// TwinCAT 3 PLC project IOLib
// ProgramVersion: 3.1.4023.0
// libraries:
//   Tc2_Standard, * (Beckhoff Automation GmbH)
//   Tc2_System, * (Beckhoff Automation GmbH)
//   Tc3_Module, * (Beckhoff Automation GmbH)
// project tree:
//   CAN/ FB_CANControl.TcPOU, ITF_CANControl.TcIO, ST_TxRxMessage.TcDUT, ST_TxRxQueue.TcDUT
//   EtherCAT/EtherCAT Devices/ DeviceInfo.TcDUT (not stored), DeviceState.TcDUT (not stored), EtherCATDeviceBase.TcPOU (not stored)
//   EtherCAT/EtherCAT Master/ EcMasterInputs.TcDUT, MasterDevState.TcDUT
//   EtherCAT/Tasks/ EcMasterConfDevices.TcPOU, EcMasterDeviceCount.TcPOU, EcMasterDeviceState.TcPOU, EcMasterFrameCount.TcPOU, EcMasterFrameStats.TcPOU, EcMasterGetAbnortalStateChange.TcPOU, EcMasterGetDeviceCRC.TcPOU, EcMasterGetDeviceId.TcPOU, EcMasterGetDeviceState.TcPOU, EcMasterProtocolError.TcPOU, EcMasterScanDevices.TcPOU, EcMasterState.TcPOU, IEcTask.TcIO, ITask.TcIO
//   EtherNetIP/ EtherNetIPDeviceBase.TcPOU, EtherNetIPMaster.TcPOU
//   Motion/RollerAxis/ EP7402_0xxx_Channel.TcPOU
//   Motion/RollerAxis/Structs/ DInputs.TcDUT, DOutputs.TcDUT, STMControl.TcDUT, STMInfoData.TcDUT, STMInputDevice.TcDUT, STMStatus.TcDUT, STMTargetVelocity.TcDUT
//   Motion/ServoAxis/ Exx72x1_DMC_Channel.TcPOU
//   Motion/ServoAxis/Structs/ DMC_Ins.TcDUT, DMC_Outs.TcDUT, DriveControl.TcDUT, DriveInputs.TcDUT, DriveOutputs.TcDUT, DriveStatus.TcDUT, PositioningControl.TcDUT, PositionStatus.TcDUT
//   Motion/StepperAxis/ Ex70x7_DMC_Channel.TcPOU
//   Motion/StepperAxis/Structs/ StartType.TcDUT, StepperENCControl.TcDUT, StepperENCStatus.TcDUT, StepperPOSControl.TcDUT, StepperPOSStatus.TcDUT, StepperSTMControl.TcDUT, StepperSTMStatus.TcDUT
//   / PlcTask.TcTTO
//   POUs/ MAIN.TcPOU
//   Profibus/ ProfibusDeviceBase.TcPOU, ProfibusMaster.TcPOU
//   ProfiNet/ ProfiNetDeviceBase.TcPOU, ProfiNetMaster.TcPOU

CONFIGURATION IOLib
    RESOURCE PLC ON TwinCAT3
        TASK PlcTask(INTERVAL := T#10ms, PRIORITY := 20);
        PROGRAM MAIN WITH PlcTask : MAIN;
    END_RESOURCE
END_CONFIGURATION

// ---- CAN/ST_TxRxMessage.TcDUT
{attribute 'pack_mode' := '1'} 
TYPE ST_TxRxMessage :
STRUCT
	dataLength : UINT;
	cobId : UDINT;
	data : ARRAY[0..7] OF BYTE;
END_STRUCT
END_TYPE

// ---- CAN/ST_TxRxQueue.TcDUT
TYPE ST_TxRxQueue :
STRUCT
	txCounter : UINT;
	rxCounter : UINT;
	noOfMessages : UINT;
	messages : ARRAY[0..9] OF ST_TxRxMessage;
END_STRUCT
END_TYPE

// ---- EtherCAT/EtherCAT Master/EcMasterInputs.TcDUT
TYPE EcMasterInputs :
STRUCT
	SlaveCount : UINT;
	DevState : UINT;
END_STRUCT
END_TYPE

// ---- EtherCAT/EtherCAT Master/MasterDevState.TcDUT
{attribute 'qualified_only'}
{attribute 'strict'}
TYPE MasterDevState :
(
	enum_member := 0
);
END_TYPE

// ---- Motion/RollerAxis/Structs/DInputs.TcDUT
TYPE DInputs :
STRUCT
	input1 : BOOL;
	input2 : BOOL;
	input3 : BOOL;
	input4 : BOOL;
	controlInput1 : BOOL;
	controlInput2 : BOOL;
	controlInput3 : BOOL;
	controlInput4 : BOOL;
END_STRUCT
END_TYPE

// ---- Motion/RollerAxis/Structs/DOutputs.TcDUT
TYPE DOutputs :
STRUCT
	output1 : BOOL;
	output2 : BOOL;
	output3 : BOOL;
	output4 : BOOL;
	controlOutput1 : BOOL;
	controlOutput2 : BOOL;
	controlOutput3 : BOOL;
	controlOutput4 : BOOL;
END_STRUCT
END_TYPE

// ---- Motion/RollerAxis/Structs/STMControl.TcDUT
TYPE STMControl :
STRUCT
	enable : BOOL;
	reset : BOOL;
	invertDirection : BOOL;
	brakeOutput : BOOL;
END_STRUCT
END_TYPE

// ---- Motion/RollerAxis/Structs/STMInfoData.TcDUT
TYPE STMInfoData :
STRUCT
	infoData1 : UINT;
	infoData2 : UINT;
	infoData3 : UINT;
END_STRUCT
END_TYPE

// ---- Motion/RollerAxis/Structs/STMInputDevice.TcDUT
TYPE STMInputDevice :
STRUCT
	deviceUnderVoltage : BOOL;
	deviceOverVoltage : BOOL;
	overTemperatureWarning : BOOL;
	overTemperatureError : BOOL;
	generalHWError : BOOL;
	chn1OpenLoad : BOOL;
	chn1ShortCircuit : BOOL;
	chn1MotorOverloadI2TWarning : BOOL;
	chn1MotorOverloadI2TError : BOOL;
	chn1AmplifierOverloadI2TWarning : BOOL;
	chn1AmplifierOverloadI2TError : BOOL;
	chn1InLimit : BOOL;
	chn1CommutationError : BOOL;
	chn2OpenLoad : BOOL;
	chn2ShortCircuit : BOOL;
	chn2MotorOverloadI2TWarning : BOOL;
	chn2MotorOverloadI2TError : BOOL;
	chn2AmplifierOverloadI2TWarning : BOOL;
	chn2AmplifierOverloadI2TError : BOOL;
	chn2InLimit : BOOL;
	chn2CommutationError : BOOL;
END_STRUCT
END_TYPE

// ---- Motion/RollerAxis/Structs/STMStatus.TcDUT
TYPE STMStatus :
STRUCT
	readyToEnable : BOOL;
	ready : BOOL;
	warning : BOOL;
	error : BOOL;
	movingPositive : BOOL;
	movingNegative : BOOL;
	txPDOToggle : BOOL;
END_STRUCT
END_TYPE

// ---- Motion/RollerAxis/Structs/STMTargetVelocity.TcDUT
TYPE STMTargetVelocity :
STRUCT
	velocity : INT;
	acceleration : UINT;
	deceleration : UINT;
END_STRUCT
END_TYPE

// ---- Motion/ServoAxis/Structs/DMC_Ins.TcDUT
TYPE DMC_Ins :
STRUCT
	DMC_Inputs : DriveInputs;
	DMC_POS_Status : PositionStatus;
	DMC_Drv_Status : DriveStatus;
END_STRUCT
END_TYPE

// ---- Motion/ServoAxis/Structs/DMC_Outs.TcDUT
TYPE DMC_Outs :
STRUCT
	DMC_DrvOuts : DriveOutputs;
	DMC_Drv_Ctrl : DriveControl;
	DMC_POS_Ctrl : PositioningControl;
END_STRUCT
END_TYPE

// ---- Motion/ServoAxis/Structs/DriveControl.TcDUT
TYPE DriveControl :
STRUCT
	Enable : BOOL;
	Reset : BOOL;
END_STRUCT
END_TYPE

// ---- Motion/ServoAxis/Structs/DriveInputs.TcDUT
TYPE DriveInputs :
STRUCT
	SetPosition : UDINT;
	SetVelocity : INT;
	ActualDriveTime : UDINT;
	ActualPositionLag : DINT;
	ActualVelocity : INT;
	ActualPosition : UDINT;
	ErrorId : UDINT;
	InputCycleCounter : USINT;
	LatchValue : UDINT;
	CyclicInfoData1 : INT;
	CyclicInforData2 : INT;
END_STRUCT
END_TYPE

// ---- Motion/ServoAxis/Structs/DriveOutputs.TcDUT
TYPE DriveOutputs :
STRUCT
	SetCounterValue : UDINT;
	TargetPosition : UDINT;
	TargetVelocity : INT;
	StartType : UINT;
	TargetAcceleration : UINT;
	TargetDeceleration : UINT;
END_STRUCT
END_TYPE

// ---- Motion/ServoAxis/Structs/DriveStatus.TcDUT
TYPE DriveStatus :
STRUCT
	ReadyToEnable : BOOL;
	Ready : BOOL;
	Warning : BOOL;
	Error : BOOL;
	MovingPositive : BOOL;
	MovingNegative : BOOL;
	DigitalInput1 : BOOL;
	DigitalInput2 : BOOL;
END_STRUCT
END_TYPE

// ---- Motion/ServoAxis/Structs/PositioningControl.TcDUT
TYPE PositioningControl :
STRUCT
	Execute : BOOL;
	EmergencyStop : BOOL;
END_STRUCT
END_TYPE

// ---- Motion/ServoAxis/Structs/PositionStatus.TcDUT
TYPE PositionStatus :
STRUCT
	Busy : BOOL;
	InTarget : BOOL;
	Warning : BOOL;
	Error : BOOL;
	Calibrated : BOOL;
	Accelerate : BOOL;
	Decelerate : BOOL;
	ReadyToExecute : BOOL;
END_STRUCT
END_TYPE

// ---- Motion/StepperAxis/Structs/StartType.TcDUT
{attribute 'qualified_only'}
{attribute 'strict'}
TYPE StartType :
(
	Absolute := 1,
	Relative := 2,
	VeloPositive := 3,
	VeloNegative := 4,
	Calibrate := 24576 
);
END_TYPE

// ---- Motion/StepperAxis/Structs/StepperENCControl.TcDUT
TYPE StepperENCControl :
STRUCT
	EnableLatchC : BOOL;
	EnableLatchPositiveEdge : BOOL;
	SetCounter : BOOL;
	EnableLatchNegativeEdge : BOOL;
	SetCounterValue : UDINT;
END_STRUCT
END_TYPE

// ---- Motion/StepperAxis/Structs/StepperENCStatus.TcDUT
TYPE StepperENCStatus :
STRUCT
	LatchCValid : BOOL;
	LatchExternalValid : BOOL;
	SetCounterDone : BOOL;
	CounterUnderflow : BOOL;
	CounterOverflow : BOOL;
	ExtrapolationStall : BOOL;
	StatusInputA : BOOL;
	StatusInputB : BOOL;
	StatusInputC : BOOL;
	StatusExternLatch : BOOL;
	SyncError : BOOL;
	TxPDOToggle : BOOL;
	CounterValue : UDINT;
	LatchValue : UDINT;
END_STRUCT
END_TYPE

// ---- Motion/StepperAxis/Structs/StepperPOSControl.TcDUT
TYPE StepperPOSControl :
STRUCT
	Execute : BOOL;
	EmergencyStop : BOOL;
	TargetPosition : UDINT;
	Velocity : INT;
	StartType : UINT;
	Acceleration : UINT;
	Deceleration : UINT;
END_STRUCT
END_TYPE

// ---- Motion/StepperAxis/Structs/StepperPOSStatus.TcDUT
TYPE StepperPOSStatus :
STRUCT
	Busy : BOOL;
	InTarget : BOOL;
	Warning : BOOL;
	Error : BOOL;
	Calibrated : BOOL;
	Accelerate : BOOL;
	Decelerate : BOOL;
	ReadyToExecute : BOOL;
	ActualPosition : UDINT;
	ActualVelocity : INT;
	ActualDriveTime : UDINT;
END_STRUCT
END_TYPE

// ---- Motion/StepperAxis/Structs/StepperSTMControl.TcDUT
TYPE StepperSTMControl :
STRUCT
	Enable : BOOL;
	Reset : BOOL;
	ReduceTorque : BOOL;
	DigitalOutput1 : BOOL;
END_STRUCT
END_TYPE

// ---- Motion/StepperAxis/Structs/StepperSTMStatus.TcDUT
TYPE StepperSTMStatus :
STRUCT
	ReadyToEnable : BOOL;
	Ready : BOOL;
	Warning : BOOL;
	Error : BOOL;
	MovingPositive : BOOL;
	MovingNegative : BOOL;
	MotorStall : BOOL;
	DigitalInput1 : BOOL;
	DigitalInput2 : BOOL;
	SyncError : BOOL;
	TxPDOToggle : BOOL;
END_STRUCT
END_TYPE

// ---- CAN/ITF_CANControl.TcIO
INTERFACE ITF_CANControl

METHOD M_GetMessage : BOOL
VAR_INPUT
END_VAR
END_METHOD

METHOD M_PushMessage : BOOL
VAR_INPUT
	messageSend : ST_TxRxMessage;
END_VAR
END_METHOD

END_INTERFACE

// ---- EtherCAT/Tasks/IEcTask.TcIO
INTERFACE IEcTask EXTENDS ITask

PROPERTY NetID : amsnetid
GET
END_GET
SET
END_SET
END_PROPERTY

END_INTERFACE

// ---- EtherCAT/Tasks/ITask.TcIO
INTERFACE ITask

METHOD Abort : BOOL
VAR_INPUT
END_VAR
END_METHOD

PROPERTY Busy : bool
GET
END_GET
END_PROPERTY

PROPERTY Done : bool
GET
END_GET
END_PROPERTY

PROPERTY Error : bool
GET
END_GET
END_PROPERTY

METHOD Execute : BOOL
VAR_INPUT
END_VAR
END_METHOD

END_INTERFACE

// ---- POUs/MAIN.TcPOU
PROGRAM MAIN
VAR
END_VAR

END_PROGRAM

// ---- CAN/FB_CANControl.TcPOU
FUNCTION_BLOCK PUBLIC FB_CANControl IMPLEMENTS ITF_CANControl
VAR_INPUT
END_VAR
VAR_OUTPUT
END_VAR
VAR
	rxQueue AT%I* : ST_TxRxQueue;
	txQueue AT%Q* : ST_TxRxQueue;
	i : INT;
	messageRecieved : ST_TxRxMessage;
END_VAR

IF rxQueue.rxCounter <> txQueue.rxCounter THEN
	//if we have recieved a message rxCounter is incremented by interface
	M_GetMessage();
END_IF

METHOD PUBLIC M_GetMessage : BOOL
VAR_INPUT
END_VAR
FOR i := 0 TO rxQueue.noOfMessages DO
	messageRecieved := rxQueue.messages[i];
END_FOR
txQueue.rxCounter := rxQueue.rxCounter;
END_METHOD

METHOD PUBLIC M_PushMessage : BOOL
VAR_INPUT
	messageSend : ST_TxRxMessage;
END_VAR
IF txQueue.txCounter = rxQueue.TxCounter THEN
	FOR i:=0 TO 1 DO
		txQueue.messages[i] := messageSend;
	End_for
	txQueue.noOfMessages := 1;
	txQueue.TxCounter := rxQueue.TxCounter + 1;
END_IF
END_METHOD

END_FUNCTION_BLOCK

// ---- EtherCAT/Tasks/EcMasterConfDevices.TcPOU
FUNCTION_BLOCK EcMasterConfDevices IMPLEMENTS IEcTask
VAR_INPUT
END_VAR
VAR_OUTPUT
END_VAR
VAR
	iState : INT;
	masterConfDevices : Tc2_EtherCAT.FB_EcGetConfSlaves;
	_confDevices : ARRAY[0..Tc2_EtherCAT.EC_MAX_SLAVES] OF Tc2_EtherCAT.ST_EcSlaveConfigData;
	_execute: BOOL;
	_done: BOOL;
	_busy: BOOL;	
	_error: BOOL;
	_netId: AMSNETID;
END_VAR

CASE iState OF
	0:
		IF _execute THEN
			_done := FALSE;
			_busy := TRUE;
			_error := FALSE;
			masterConfDevices.bExecute := TRUE;
			IF masterConfDevices.bBusy THEN
				iState := 10;
				_execute := FALSE;
			END_IF
		END_IF
	10:
		IF NOT masterConfDevices.bBusy THEN
			IF NOT masterConfDevices.bError THEN
				_done := TRUE;
			ELSE
				_error := TRUE;
			END_IF
			_busy := FALSE;
			masterConfDevices.bExecute := FALSE;
			iState := 0;
		END_IF
END_CASE

masterConfDevices(sNetId := Tc2_System.F_CreateAmsNetId(nIds := NetId), 
					pArrEcConfSlaveInfo := ADR(_confDevices), 
					cbBufLen := SIZEOF(_confDevices));

{warning 'add method implementation '}
METHOD Abort : BOOL
masterConfDevices.bExecute := FALSE;
_busy := FALSE;
_execute := FALSE;
Abort := TRUE;
iState := 0;
END_METHOD

{warning 'add property implementation'}
PROPERTY Busy : BOOL
GET
Busy := _busy;
END_GET
END_PROPERTY

PROPERTY ConfiguredDevices : reference to array[0..Ec_Max_slaves] of St_ecslaveconfigdata
GET
ConfiguredDevices REF= _confDevices;
END_GET
END_PROPERTY

{warning 'add property implementation'}
PROPERTY Done : BOOL
GET
Done := _done;
END_GET
END_PROPERTY

{warning 'add property implementation'}
PROPERTY Error : BOOL
GET
Error := _error;
END_GET
END_PROPERTY

{warning 'add method implementation '}
METHOD Execute : BOOL
IF NOT masterConfDevices.bBusy THEN
	Execute := _execute := true;
END_IF
END_METHOD

{warning 'add property implementation'}
PROPERTY NetID : amsnetid
GET
NetID := _netId;
END_GET
SET
_netId := NetID;
END_SET
END_PROPERTY

PROPERTY NumberConfDevices : udint
GET
NumberConfDevices := masterConfDevices.nSlaves;
END_GET
END_PROPERTY

END_FUNCTION_BLOCK

// ---- EtherCAT/Tasks/EcMasterDeviceCount.TcPOU
FUNCTION_BLOCK PUBLIC EcMasterDeviceCount IMPLEMENTS IEcTask
VAR_INPUT
END_VAR
VAR_OUTPUT
END_VAR
VAR
	iState : INT;
	masterDeviceCount : Tc2_EtherCAT.FB_EcGetSlaveCount;
	_execute: BOOL;
	_done: BOOL;
	_busy: BOOL;
	_error: BOOL;
	_netId: AMSNETID;
END_VAR

CASE iState OF
	0:
		IF _execute THEN
			_done := FALSE;
			_busy := TRUE;
			_error := FALSE;
			masterDeviceCount.bExecute := TRUE;
			IF masterDeviceCount.bBusy THEN
				iState := 10;
				_execute := false;
			END_IF
		END_IF
	10:
		IF NOT masterDeviceCount.bBusy THEN
			IF NOT masterDeviceCount.bError THEN
				_done := TRUE;
			ELSE
				_error := TRUE;
			END_IF
			_busy := FALSE;
			masterDeviceCount.bExecute := FALSE;
			iState := 0;
		END_IF
END_CASE

masterDeviceCount(sNetId := Tc2_System.F_CreateAmsNetId(nIds := NetId));

{warning 'add method implementation '}
METHOD Abort : BOOL
masterDeviceCount.bExecute := FALSE;
_busy := FALSE;
_execute := FALSE;
Abort := TRUE;
iState := 0;
END_METHOD

{warning 'add property implementation'}
PROPERTY Busy : BOOL
GET
Busy := _busy;
END_GET
END_PROPERTY

{warning 'add property implementation'}
PROPERTY Done : BOOL
GET
Done := _done;
END_GET
END_PROPERTY

{warning 'add property implementation'}
PROPERTY Error : BOOL
GET
Error := _error;
END_GET
END_PROPERTY

METHOD Execute : BOOL
VAR_INPUT
END_VAR
IF NOT Busy THEN
	Execute := _execute := TRUE;
END_IF
END_METHOD

{warning 'add property implementation'}
PROPERTY NetID : amsnetid
GET
NetID := _netId;
END_GET
SET
_netId := NetID;
END_SET
END_PROPERTY

PROPERTY NumberDevices : uint
GET
NumberDevices := masterDeviceCount.nSlaves;
END_GET
END_PROPERTY

END_FUNCTION_BLOCK

// ---- EtherCAT/Tasks/EcMasterDeviceState.TcPOU
FUNCTION_BLOCK EcMasterDeviceState IMPLEMENTS IEcTask
VAR_INPUT
END_VAR
VAR_OUTPUT
END_VAR
VAR
	iState : INT;
	masterDeviceState : Tc2_EtherCAT.FB_EcGetMasterDevState;
	_execute: BOOL;
	_done: BOOL;
	_busy: BOOL;
	_error: BOOL;
	_netId: AMSNETID;
END_VAR

CASE iState OF
	0:
		IF _execute THEN
			_done := FALSE;
			_busy := TRUE;
			_error := FALSE;
			masterDeviceState.bExecute := TRUE;
			IF masterDeviceState.bBusy THEN
				iState := 10;
				_execute := false;
			END_IF
		END_IF
	10:
		IF NOT masterDeviceState.bBusy THEN
			IF NOT masterDeviceState.bError THEN
				_done := TRUE;
			ELSE
				_error := TRUE;
			END_IF
			_busy := FALSE;
			masterDeviceState.bExecute := FALSE;
			iState := 0;
		END_IF
END_CASE

masterDeviceState(sNetId := Tc2_System.F_CreateAmsNetId(nIds := NetId));

{warning 'add method implementation '}
METHOD Abort : BOOL
masterDeviceState.bExecute := FALSE;
_busy := FALSE;
_execute := FALSE;
Abort := TRUE;
iState := 0;
END_METHOD

{warning 'add property implementation'}
PROPERTY Busy : BOOL
GET
Busy := _busy;
END_GET
END_PROPERTY

{warning 'add property implementation'}
PROPERTY Done : BOOL
GET
Done := _done;
END_GET
END_PROPERTY

{warning 'add property implementation'}
PROPERTY Error : BOOL
GET
Error := _error;
END_GET
END_PROPERTY

{warning 'add method implementation '}
METHOD Execute : BOOL
IF NOT masterDeviceState.bBusy THEN
	Execute := _execute := true;
END_IF
END_METHOD

PROPERTY MasterDevState : word
GET
MasterDevState := masterDeviceState.nDevState;
END_GET
END_PROPERTY

{warning 'add property implementation'}
PROPERTY NetID : amsnetid
GET
NetID := _netId;
END_GET
SET
_netId := NetID;
END_SET
END_PROPERTY

END_FUNCTION_BLOCK

// ---- EtherCAT/Tasks/EcMasterFrameCount.TcPOU
FUNCTION_BLOCK EcMasterFrameCount IMPLEMENTS IEcTask
VAR_INPUT
END_VAR
VAR_OUTPUT
END_VAR
VAR
	iState : INT;
	masterFrameCount : Tc2_EtherCAT.FB_EcMasterFrameCount;
	_execute: BOOL;
	_done: BOOL;
	_busy: BOOL;
	_error: BOOL;
	_netId: AMSNETID;
END_VAR

CASE iState OF
	0:
		IF _execute THEN
			_done := FALSE;
			_busy := TRUE;
			_error := FALSE;
			masterFrameCount.bExecute := TRUE;
			IF masterFrameCount.bBusy THEN
				iState := 10;
				_execute := false;
			END_IF
		END_IF
	10:
		IF NOT masterFrameCount.bBusy THEN
			IF NOT masterFrameCount.bError THEN
				_done := TRUE;
			ELSE
				_error := TRUE;
			END_IF
			_busy := FALSE;
			masterFrameCount.bExecute := FALSE;
			iState := 0;
		END_IF
END_CASE

masterFrameCount(sNetId := Tc2_System.F_CreateAmsNetId(nIds := NetId));

{warning 'add method implementation '}
METHOD Abort : BOOL
masterFrameCount.bExecute := FALSE;
_busy := FALSE;
_execute := FALSE;
Abort := TRUE;
iState := 0;
END_METHOD

{warning 'add property implementation'}
PROPERTY Busy : BOOL
GET
Busy := _busy;
END_GET
END_PROPERTY

{warning 'add property implementation'}
PROPERTY Done : BOOL
GET
Done := _done;
END_GET
END_PROPERTY

{warning 'add property implementation'}
PROPERTY Error : BOOL
GET
Error := _error;
END_GET
END_PROPERTY

{warning 'add method implementation '}
METHOD Execute : BOOL
IF NOT masterFrameCount.bBusy THEN
	Execute := _execute := True;
END_IF
END_METHOD

PROPERTY FrameNumber : UDINT
GET
FrameNumber := masterFrameCount.nFrames;
END_GET
END_PROPERTY

{warning 'add property implementation'}
PROPERTY NetID : amsnetid
GET
NetID := _netId;
END_GET
SET
_netId := NetID;
END_SET
END_PROPERTY

END_FUNCTION_BLOCK

// ---- EtherCAT/Tasks/EcMasterFrameStats.TcPOU
FUNCTION_BLOCK PUBLIC EcMasterFrameStats IMPLEMENTS IEcTask
VAR_INPUT
END_VAR
VAR_OUTPUT
END_VAR
VAR
	iState : INT;
	masterFrameStats : Tc2_EtherCAT.FB_EcMasterFrameStatistic;
	_execute: BOOL;
	_done: BOOL;
	_busy: BOOL;
	_error: BOOL;
	_netId: AMSNETID;
END_VAR

CASE iState OF
	0:
		IF _execute THEN
			_done := FALSE;
			_busy := TRUE;
			_error := FALSE;
			masterFrameStats.bExecute := TRUE;
			IF masterFrameStats.bBusy THEN
				iState := 10;
				_execute := false;
			END_IF
		END_IF
	10:
		IF NOT masterFrameStats.bBusy THEN
			IF NOT masterFrameStats.bError THEN
				_done := TRUE;
			ELSE
				_error := TRUE;
			END_IF
			_busy := FALSE;
			masterFrameStats.bExecute := FALSE;
			iState := 0;
		END_IF
END_CASE

masterFrameStats(sNetId := Tc2_System.F_CreateAmsNetId(nIds := NetId));

{warning 'add method implementation '}
METHOD Abort : BOOL
masterFrameStats.bExecute := FALSE;
_busy := FALSE;
_execute := FALSE;
Abort := TRUE;
iState := 0;
END_METHOD

{warning 'add property implementation'}
PROPERTY Busy : BOOL
GET
Busy := _busy;
END_GET
END_PROPERTY

{warning 'add property implementation'}
PROPERTY Done : BOOL
GET
Done := _done;
END_GET
END_PROPERTY

{warning 'add property implementation'}
PROPERTY Error : BOOL
GET
Error := _error;
END_GET
END_PROPERTY

METHOD Execute : BOOL
VAR_INPUT
END_VAR
IF NOT Busy THEN
	Execute := _execute := TRUE;
END_IF
END_METHOD

PROPERTY FramesPerSecond  : LREAL
GET
FramesPerSecond := masterFrameStats.fFramesPerSecond;
END_GET
END_PROPERTY

PROPERTY LostFrames : UDINT
GET
LostFrames := masterFrameStats.nLostFrames;
END_GET
END_PROPERTY

PROPERTY LostQueuedFrames : udint
GET
LostQueuedFrames := masterFrameStats.nLostQueuedFrames;
END_GET
END_PROPERTY

{warning 'add property implementation'}
PROPERTY NetID : amsnetid
GET
NetID := _netId;
END_GET
SET
_netId := NetID;
END_SET
END_PROPERTY

PROPERTY QueuedFramesPerSecond : lreal
GET
QueuedFramesPerSecond := masterFrameStats.fQueuedFramesPerSecond;
END_GET
END_PROPERTY

END_FUNCTION_BLOCK

// ---- EtherCAT/Tasks/EcMasterGetAbnortalStateChange.TcPOU
FUNCTION_BLOCK EcMasterGetAbnortalStateChange IMPLEMENTS IEcTask
VAR_INPUT
END_VAR
VAR_OUTPUT
END_VAR
VAR
	iState : INT;
	masterAbnormalStateChanges : Tc2_EtherCAT.FB_EcGetAllSlaveAbnormalStateChanges;
	_abnormalStates : ARRAY[0..Tc2_EtherCAT.EC_MAX_SLAVES] OF UDINT;
	_execute: BOOL;
	_done: BOOL;
	_busy: BOOL;
	_error: BOOL;
	_netId: AMSNETID;
END_VAR

CASE iState OF
	0:
		IF _execute THEN
			_done := FALSE;
			_busy := TRUE;
			_error := FALSE;
			masterAbnormalStateChanges.bExecute := TRUE;
			IF masterAbnormalStateChanges.bBusy THEN
				iState := 10;
				_execute := false;
			END_IF
		END_IF
	10:
		IF NOT masterAbnormalStateChanges.bBusy THEN
			IF NOT masterAbnormalStateChanges.bError THEN
				_done := TRUE;
			ELSE
				_error := TRUE;
			END_IF
			_busy := FALSE;
			masterAbnormalStateChanges.bExecute := FALSE;
			iState := 0;
		END_IF
END_CASE

masterAbnormalStateChanges(sNetId := Tc2_System.F_CreateAmsNetId(nIds := NetId),
							pAddrBuf := ADR(_abnormalStates),
							cbBufLen := SIZEOF(_abnormalStates));

PROPERTY AbnormalStateChanges : reference to array[0..EC_MAX_Slaves] of udint
GET
AbnormalStateChanges REF= _abnormalStates;
END_GET
END_PROPERTY

{warning 'add method implementation '}
METHOD Abort : BOOL
masterAbnormalStateChanges.bExecute := FALSE;
_busy := FALSE;
_execute := FALSE;
Abort := TRUE;
iState := 0;
END_METHOD

{warning 'add property implementation'}
PROPERTY Busy : BOOL
GET
Busy := _busy;
END_GET
END_PROPERTY

{warning 'add property implementation'}
PROPERTY Done : BOOL
GET
Done := _done;
END_GET
END_PROPERTY

{warning 'add property implementation'}
PROPERTY Error : BOOL
GET
Error := _error;
END_GET
END_PROPERTY

{warning 'add method implementation '}
METHOD Execute : BOOL
IF NOT masterAbnormalStateChanges.bBusy THEN
	Execute := _execute := true;
END_IF
END_METHOD

{warning 'add property implementation'}
PROPERTY NetID : amsnetid
GET
NetID := _netId;
END_GET
SET
_netId := NetID;
END_SET
END_PROPERTY

END_FUNCTION_BLOCK

// ---- EtherCAT/Tasks/EcMasterGetDeviceCRC.TcPOU
FUNCTION_BLOCK EcMasterGetDeviceCRC IMPLEMENTS IEcTask
VAR_INPUT
END_VAR
VAR_OUTPUT
END_VAR
VAR
	iState : INT;
	getDeviceCRC : Tc2_EtherCAT.FB_EcGetSlaveCrcErrorEx;
	_execute: BOOL;
	_done: BOOL;
	_busy: BOOL;
	_error: BOOL;
	_netId: AMSNETID;
END_VAR

CASE iState OF
	0:
		IF _execute THEN
			_done := FALSE;
			_busy := TRUE;
			_error := FALSE;
			getDeviceCRC.bExecute := TRUE;
			IF getDeviceCRC.bBusy THEN
				iState := 10;
				_execute := false;
			END_IF
		END_IF
	10:
		IF NOT getDeviceCRC.bBusy THEN
			IF NOT getDeviceCRC.bError THEN
				_done := TRUE;
			ELSE
				_error := TRUE;
			END_IF
			_busy := FALSE;
			getDeviceCRC.bExecute := FALSE;
			iState := 0;
		END_IF
END_CASE

getDeviceCRC(sNetId := Tc2_System.F_CreateAmsNetId(nIds := NetId));

{warning 'add method implementation '}
METHOD Abort : BOOL
getDeviceCRC.bExecute := FALSE;
_busy := FALSE;
_execute := FALSE;
Abort := TRUE;
iState := 0;
END_METHOD

{warning 'add property implementation'}
PROPERTY Busy : BOOL
GET
Busy := _busy;
END_GET
END_PROPERTY

PROPERTY DeviceAddr : uint
GET
DeviceAddr := getDeviceCRC.nSlaveAddr;
END_GET
SET
getDeviceCRC.nSlaveAddr := DeviceAddr;
END_SET
END_PROPERTY

PROPERTY DeviceCRC :  ST_EcCrcErrorEx
GET
DeviceCRC := getDeviceCRC.crcError;
END_GET
END_PROPERTY

{warning 'add property implementation'}
PROPERTY Done : BOOL
GET
Done := _done;
END_GET
END_PROPERTY

{warning 'add property implementation'}
PROPERTY Error : BOOL
GET
Error := _error;
END_GET
END_PROPERTY

{warning 'add method implementation '}
METHOD Execute : BOOL
IF NOT getDeviceCRC.bBusy THEN
	Execute := _execute := true;
END_IF
END_METHOD

{warning 'add property implementation'}
PROPERTY NetID : amsnetid
GET
NetID := _netId;
END_GET
SET
_netId := NetID;
END_SET
END_PROPERTY

END_FUNCTION_BLOCK

// ---- EtherCAT/Tasks/EcMasterGetDeviceId.TcPOU
FUNCTION_BLOCK EcMasterGetDeviceId IMPLEMENTS IEcTask
VAR_INPUT
END_VAR
VAR_OUTPUT
END_VAR
VAR
	iState : INT;
	getDeviceIdentity : Tc2_EtherCAT.FB_EcGetSlaveIdentity;
	_execute: BOOL;
	_done: BOOL;
	_busy: BOOL;
	_error: BOOL;
	_netId: AMSNETID;
END_VAR

CASE iState OF
	0:
		IF _execute THEN
			_done := FALSE;
			_busy := TRUE;
			_error := FALSE;
			getDeviceIdentity.bExecute := TRUE;
			IF getDeviceIdentity.bBusy THEN
				iState := 10;
				_execute := false;
			END_IF
		END_IF
	10:
		IF NOT getDeviceIdentity.bBusy THEN
			IF NOT getDeviceIdentity.bError THEN
				_done := TRUE;
			ELSE
				_error := TRUE;
			END_IF
			_busy := FALSE;
			getDeviceIdentity.bExecute := FALSE;
			iState := 0;
		END_IF
END_CASE

getDeviceIdentity(sNetId := Tc2_System.F_CreateAmsNetId(nIds := NetId));

{warning 'add method implementation '}
METHOD Abort : BOOL
getDeviceIdentity.bExecute := FALSE;
_busy := FALSE;
_execute := FALSE;
Abort := TRUE;
iState := 0;
END_METHOD

{warning 'add property implementation'}
PROPERTY Busy : BOOL
GET
Busy := _busy;
END_GET
END_PROPERTY

PROPERTY DeviceAddr : uint
GET
DeviceAddr := getDeviceIdentity.nSlaveAddr;
END_GET
SET
getDeviceIdentity.nSlaveAddr := DeviceAddr;
END_SET
END_PROPERTY

PROPERTY DeviceIdentity : ST_EcSlaveIdentity
GET
DeviceIdentity := getDeviceIdentity.identity;
END_GET
END_PROPERTY

{warning 'add property implementation'}
PROPERTY Done : BOOL
GET
Done := _done;
END_GET
END_PROPERTY

{warning 'add property implementation'}
PROPERTY Error : BOOL
GET
Error := _error;
END_GET
END_PROPERTY

{warning 'add method implementation '}
METHOD Execute : BOOL
IF NOT getDeviceIdentity.bBusy THEN
	Execute := _execute := true;
END_IF
END_METHOD

{warning 'add property implementation'}
PROPERTY NetID : amsnetid
GET
NetID := _netId;
END_GET
SET
_netId := NetID;
END_SET
END_PROPERTY

END_FUNCTION_BLOCK

// ---- EtherCAT/Tasks/EcMasterGetDeviceState.TcPOU
FUNCTION_BLOCK EcMasterGetDeviceState IMPLEMENTS IEcTask
VAR_INPUT
END_VAR
VAR_OUTPUT
END_VAR
VAR
	iState : INT;
	getDeviceState : Tc2_EtherCAT.FB_EcGetSlaveState;
	_execute: BOOL;
	_done: BOOL;
	_busy: BOOL;
	_error: BOOL;
	_netId: AMSNETID;
END_VAR

CASE iState OF
	0:
		IF _execute THEN
			_done := FALSE;
			_busy := TRUE;
			_error := FALSE;
			getDeviceState.bExecute := TRUE;
			IF getDeviceState.bBusy THEN
				iState := 10;
				_execute := false;
			END_IF
		END_IF
	10:
		IF NOT getDeviceState.bBusy THEN
			IF NOT getDeviceState.bError THEN
				_done := TRUE;
			ELSE
				_error := TRUE;
			END_IF
			_busy := FALSE;
			getDeviceState.bExecute := FALSE;
			iState := 0;
		END_IF
END_CASE

getDeviceState(sNetId := Tc2_System.F_CreateAmsNetId(nIds := NetId));

{warning 'add method implementation '}
METHOD Abort : BOOL
getDeviceState.bExecute := FALSE;
_busy := FALSE;
_execute := FALSE;
Abort := TRUE;
iState := 0;
END_METHOD

{warning 'add property implementation'}
PROPERTY Busy : BOOL
GET
Busy := _busy;
END_GET
END_PROPERTY

PROPERTY DeviceAddr : uint
GET
DeviceAddr := getDeviceState.nSlaveAddr;
END_GET
SET
getDeviceState.nSlaveAddr := DeviceAddr;
END_SET
END_PROPERTY

PROPERTY DeviceState : ST_EcSlaveState
GET
DeviceState := getDeviceState.state;
END_GET
END_PROPERTY

{warning 'add property implementation'}
PROPERTY Done : BOOL
GET
Done := _done;
END_GET
END_PROPERTY

{warning 'add property implementation'}
PROPERTY Error : BOOL
GET
Error := _error;
END_GET
END_PROPERTY

{warning 'add method implementation '}
METHOD Execute : BOOL
IF NOT getDeviceState.bBusy THEN
	Execute := _execute := true;
END_IF
END_METHOD

{warning 'add property implementation'}
PROPERTY NetID : amsnetid
GET
NetID := _netId;
END_GET
SET
_netId := NetID;
END_SET
END_PROPERTY

END_FUNCTION_BLOCK

// ---- EtherCAT/Tasks/EcMasterProtocolError.TcPOU
FUNCTION_BLOCK EcMasterProtocolError IMPLEMENTS IEcTask
VAR_INPUT
END_VAR
VAR_OUTPUT
END_VAR
VAR
	iState : INT;
	masterProtocolErr : Tc2_EtherCAT.FB_EcGetLastProtErrInfo;
	_execute: BOOL;
	_done: BOOL;
	_busy: BOOL;
	_error: BOOL;
	_netId: AMSNETID;
END_VAR

CASE iState OF
	0:
		IF _execute THEN
			_done := FALSE;
			_busy := TRUE;
			_error := FALSE;
			masterProtocolErr.bExecute := TRUE;
			IF masterProtocolErr.bBusy THEN
				iState := 10;
				_execute := false;
			END_IF
		END_IF
	10:
		IF NOT masterProtocolErr.bBusy THEN
			IF NOT masterProtocolErr.bError THEN
				_done := TRUE;
			ELSE
				_error := TRUE;
			END_IF
			_busy := FALSE;
			masterProtocolErr.bExecute := FALSE;
			iState := 0;
		END_IF
END_CASE

masterProtocolErr(sNetId := Tc2_System.F_CreateAmsNetId(nIds := NetId));

{warning 'add method implementation '}
METHOD Abort : BOOL
masterProtocolErr.bExecute := FALSE;
_busy := FALSE;
_execute := FALSE;
Abort := TRUE;
iState := 0;
END_METHOD

{warning 'add property implementation'}
PROPERTY Busy : BOOL
GET
Busy := _busy;
END_GET
END_PROPERTY

PROPERTY DeviceAddr : uint
GET
DeviceAddr := masterProtocolErr.nSlaveAddr;
END_GET
SET
masterProtocolErr.nSlaveAddr := DeviceAddr;
END_SET
END_PROPERTY

{warning 'add property implementation'}
PROPERTY Done : BOOL
GET
Done := _done;
END_GET
END_PROPERTY

{warning 'add property implementation'}
PROPERTY Error : BOOL
GET
Error := _error;
END_GET
END_PROPERTY

{warning 'add method implementation '}
METHOD Execute : BOOL
IF NOT masterProtocolErr.bBusy THEN
	Execute := _execute := TRUE;
END_IF
END_METHOD

PROPERTY LastProtocolError : ST_EcLastProtErrInfo
GET
LastProtocolError := masterProtocolErr.info;
END_GET
END_PROPERTY

{warning 'add property implementation'}
PROPERTY NetID : amsnetid
GET
NetID := _netId;
END_GET
SET
_netId := NetID;
END_SET
END_PROPERTY

PROPERTY ProtocolType : E_EcMbxProtType
GET
ProtocolType := masterProtocolErr.eProtocol;
END_GET
SET
masterProtocolErr.eProtocol := ProtocolType;
END_SET
END_PROPERTY

END_FUNCTION_BLOCK

// ---- EtherCAT/Tasks/EcMasterScanDevices.TcPOU
FUNCTION_BLOCK EcMasterScanDevices IMPLEMENTS IEcTask
VAR_INPUT
END_VAR
VAR_OUTPUT
END_VAR
VAR
	iState : INT;
	masterScanDevices : Tc2_EtherCAT.FB_EcGetScannedSlaves;
	_scanDevices : ARRAY[0..Tc2_EtherCAT.EC_MAX_SLAVES] OF Tc2_EtherCAT.ST_EcSlaveScannedData;
	_execute: BOOL;
	_done: BOOL;
	_busy: BOOL;
	_error: BOOL;
	_netId: AMSNETID;
END_VAR

CASE iState OF
	0:
		IF _execute THEN
			_done := FALSE;
			_busy := TRUE;
			_error := FALSE;
			masterScanDevices.bExecute := TRUE;
			IF masterScanDevices.bBusy THEN
				iState := 10;
				_execute := false;
			END_IF
		END_IF
	10:
		IF NOT masterScanDevices.bBusy THEN
			IF NOT masterScanDevices.bError THEN
				_done := TRUE;
			ELSE
				_error := TRUE;
			END_IF
			_busy := FALSE;
			masterScanDevices.bExecute := FALSE;
			iState := 0;
		END_IF
END_CASE

masterScanDevices(sNetId := Tc2_System.F_CreateAmsNetId(nIds := NetId), 
					pArrEcScannedSlaveInfo := ADR(_scanDevices), 
					cbBufLen := SIZEOF(_scanDevices));

{warning 'add method implementation '}
METHOD Abort : BOOL
masterScanDevices.bExecute := FALSE;
_busy := FALSE;
_execute := FALSE;
Abort := TRUE;
iState := 0;
END_METHOD

{warning 'add property implementation'}
PROPERTY Busy : BOOL
GET
Busy := _busy;
END_GET
END_PROPERTY

{warning 'add property implementation'}
PROPERTY Done : BOOL
GET
Done := _done;
END_GET
END_PROPERTY

{warning 'add property implementation'}
PROPERTY Error : BOOL
GET
Error := _error;
END_GET
END_PROPERTY

{warning 'add method implementation '}
METHOD Execute : BOOL
IF NOT masterScanDevices.bBusy THEN
	Execute := _execute := true;
END_IF
END_METHOD

{warning 'add property implementation'}
PROPERTY NetID : amsnetid
GET
NetID := _netId;
END_GET
SET
_netId := NetID;
END_SET
END_PROPERTY

PROPERTY NumberScanDevices : udint
GET
NumberScanDevices := masterScanDevices.nSlaves;
END_GET
END_PROPERTY

PROPERTY ScannedDevices : reference to array[0..EC_MAX_Slaves] of ST_EcSlaveScannedData
GET
ScannedDevices REF= _scanDevices;
END_GET
END_PROPERTY

END_FUNCTION_BLOCK

// ---- EtherCAT/Tasks/EcMasterState.TcPOU
{attribute 'hide_all_locals'}
FUNCTION_BLOCK EcMasterState IMPLEMENTS IEcTask
VAR_INPUT
END_VAR
VAR_OUTPUT
END_VAR
VAR
	iState : INT;
	getMasterState : Tc2_EtherCAT.FB_EcGetMasterState;
	_execute: BOOL;
	_done: BOOL;
	_busy: BOOL;
	_error: BOOL;
	
END_VAR

CASE iState OF
	0:
		IF _execute THEN
			_done := FALSE;
			_busy := TRUE;
			_error := FALSE;
			getMasterState.bExecute := TRUE;
			IF getMasterState.bBusy THEN
				iState := 10;
				_execute := false;
			END_IF
		END_IF
	10:
		IF NOT getMasterState.bBusy THEN
			IF NOT getMasterState.bError THEN
				_done := TRUE;
			ELSE
				_error := TRUE;
			END_IF
			_busy := FALSE;
			getMasterState.bExecute := FALSE;
			iState := 0;
		END_IF
END_CASE

getMasterState(sNetId := Tc2_System.F_CreateAmsNetId(nIds := NetId));

{warning 'add method implementation '}
METHOD Abort : BOOL
getMasterState.bExecute := FALSE;
_busy := FALSE;
_execute := FALSE;
Abort := TRUE;
iState := 0;
END_METHOD

{warning 'add property implementation'}
PROPERTY Busy : BOOL
GET
Busy := _busy;
END_GET
END_PROPERTY

{warning 'add property implementation'}
PROPERTY Done : BOOL
GET
Done := _done;
END_GET
END_PROPERTY

{warning 'add property implementation'}
PROPERTY Error : BOOL
GET
Error := _error;
END_GET
END_PROPERTY

{warning 'add method implementation '}
METHOD Execute : BOOL
IF NOT getMasterState.bBusy THEN
	Execute := _execute := TRUE;
END_IF
END_METHOD

PROPERTY MasterState : word
GET
MasterState := getMasterState.state;
END_GET
END_PROPERTY

{warning 'add property implementation'}
PROPERTY NetID : amsnetid
GET
NetID := _netId;
END_GET
SET
_netId := NetID;
END_SET
END_PROPERTY

END_FUNCTION_BLOCK

// ---- EtherNetIP/EtherNetIPDeviceBase.TcPOU
FUNCTION_BLOCK EtherNetIPDeviceBase
VAR_INPUT
END_VAR
VAR_OUTPUT
END_VAR
VAR
	State AT%i* : UINT;
END_VAR

END_FUNCTION_BLOCK

// ---- EtherNetIP/EtherNetIPMaster.TcPOU
FUNCTION_BLOCK EtherNetIPMaster
VAR_INPUT
END_VAR
VAR_OUTPUT
END_VAR
VAR
	DevState AT%i* : UINT;
END_VAR

END_FUNCTION_BLOCK

// ---- Motion/RollerAxis/EP7402_0xxx_Channel.TcPOU
FUNCTION_BLOCK EP7402_0xxx_Channel
VAR_INPUT
END_VAR
VAR_OUTPUT
END_VAR
VAR
	DI_Inputs AT%I* : DInputs;
	DO_Outputs AT%Q* : DOutputs;
	STM_Control AT%Q* : STMControl;
	STM_Info_data AT%I* : STMInfoData;
	STM_Input_Device AT%I* : STMInputDevice;
	STM_Status AT%I* : STMStatus;
	STM_Target_Velocity AT%Q* : STMTargetVelocity;
	
	_acceleration : UINT := 100;
	_deceleration : UINT := 100;
	
	State :(
		_00_mWait,
        _01_mReset,
        _02_mEnable,
		_03_mStop,
		_04_RunAtVelo,
		_05_mDisable);
		
	tonHoldHigh	: ton;
		
END_VAR

CASE State OF
        _00_mWait : 
			;
        _01_mReset : 
			STM_Control.reset := TRUE;
			tonHoldHigh(in := TRUE, pt := T#500MS);
			IF tonHoldHigh.Q THEN
				STM_Control.reset := FALSE;
				IF STM_Status.error = FALSE AND
					STM_Status.warning = FALSE AND
					STM_Status.ready = TRUE
				THEN
					State := _00_mWait;
					tonHoldHigh(in := FALSE);
				END_IF
			END_IF
			
        _02_mEnable : 
			IF STM_Status.error THEN				
				State := _01_mReset;
			ELSE
				STM_Control.enable := TRUE;			
			END_IF

			
		_04_RunAtVelo :
			;
			
		_03_mStop : 
			STM_Target_Velocity.velocity := 0;
			IF STM_Status.ready THEN	
				State := _02_mEnable;
			END_IF
			
		_05_mDisable:
			STM_Control.enable := FALSE;
			State := _00_mWait;
		
			
END_CASE

PROPERTY PUBLIC Acceleration : uint
GET
Acceleration := _acceleration;
END_GET
SET
_acceleration := Acceleration;
END_SET
END_PROPERTY

PROPERTY PUBLIC Deceleration : uint
GET
Deceleration := _deceleration;
END_GET
SET
_deceleration := Deceleration;
END_SET
END_PROPERTY

METHOD Disable : BOOL
VAR_INPUT
END_VAR
IF STM_Status.ready THEN
	State := _05_mDisable;
END_IF
END_METHOD

METHOD Enable : BOOL
VAR_INPUT
END_VAR
IF STM_Status.readyToEnable THEN
	State := _02_mEnable;
END_IF
END_METHOD

METHOD MoveNeg : BOOL
VAR_INPUT
END_VAR
STM_Control.invertDirection := TRUE;
STM_Target_Velocity.velocity := 6000;
STM_Target_Velocity.acceleration := _acceleration;
STM_Target_Velocity.deceleration := _deceleration;
State := _04_RunAtVelo;
END_METHOD

METHOD MovePos : BOOL
VAR_INPUT
END_VAR
STM_Control.invertDirection := FALSE;
STM_Target_Velocity.velocity := 6000;
STM_Target_Velocity.acceleration := _acceleration;
STM_Target_Velocity.deceleration := _deceleration;
State := _04_RunAtVelo;
END_METHOD

METHOD Reset : BOOL
VAR_INPUT
END_VAR
IF STM_Status.error OR STM_Status.warning THEN
	State := _01_mReset;
END_IF
END_METHOD

METHOD Stop : BOOL
VAR_INPUT
END_VAR
IF STM_Status.movingNegative OR STM_Status.movingPositive THEN
	State := _03_mStop;
END_IF
END_METHOD

END_FUNCTION_BLOCK

// ---- Motion/ServoAxis/Exx72x1_DMC_Channel.TcPOU
FUNCTION_BLOCK Exx72x1_DMC_Channel
VAR_INPUT
END_VAR
VAR_OUTPUT
END_VAR
VAR
	//Properties
	_acceleration : UINT := 4000; 	//default to 4s accel
	_deceleration : UINT := 4000;	//default to 4s decel
	_startType : UINT := 1; 		//default to abs moves
	_scale : REAL := 360; 			//default to 360 degree scale factor
	
	//Locals
	dmc_inputs AT%I* : DMC_Ins;
	dmc_outputs AT%q* : DMC_Outs;
	xMove: BOOL;
	iMove: INT;
	
	posDemand : REAL;
	currentPos : REAL;
END_VAR

MoveSequence();

dmc_outputs.DMC_DrvOuts.TargetPosition := REAL_TO_UDINT(posDemand * (1048576/360));
currentPos := UDINT_TO_REAL( dmc_inputs.DMC_Inputs.ActualPosition)*(360.0/1048576.0);

PROPERTY PUBLIC Acceleration : uint
GET
Acceleration := _acceleration;
END_GET
SET
_acceleration := Acceleration;
END_SET
END_PROPERTY

PROPERTY PUBLIC Deceleration : uint
GET
Deceleration := _deceleration;
END_GET
SET
_deceleration := Deceleration;
END_SET
END_PROPERTY

METHOD PUBLIC Enable : BOOL
VAR_INPUT
END_VAR
IF dmc_inputs.DMC_Drv_Status.ReadyToEnable THEN
	dmc_outputs.DMC_Drv_Ctrl.Enable := TRUE;
END_IF
END_METHOD

PROPERTY PUBLIC Enabled : bool
GET
Enabled := dmc_inputs.DMC_Drv_Status.Ready AND dmc_inputs.DMC_POS_Status.ReadyToExecute;
END_GET
END_PROPERTY

PROPERTY PUBLIC Error : bool
GET
Error := dmc_inputs.DMC_Drv_Status.Error;
END_GET
END_PROPERTY

METHOD PUBLIC MoveAxis : BOOL
VAR_INPUT
	PositioningControl : real;
	Velocity : INT;
END_VAR
dmc_outputs.DMC_DrvOuts.TargetPosition := REAL_TO_UDINT(PositioningControl*(1048576/_scale));
dmc_outputs.DMC_DrvOuts.TargetVelocity := Velocity;
dmc_outputs.DMC_DrvOuts.StartType := _startType;
dmc_outputs.DMC_DrvOuts.TargetAcceleration := _acceleration;
dmc_outputs.DMC_DrvOuts.TargetDeceleration := _deceleration;
xMove := TRUE;
MoveAxis := TRUE;
END_METHOD

METHOD PRIVATE MoveSequence : BOOL
VAR_INPUT
END_VAR
CASE iMove OF 
	0: 
		IF dmc_inputs.DMC_POS_Status.ReadyToExecute AND xMove THEN
			xMove := FALSE;
			iMove := 10;
		END_IF
	10:
		dmc_outputs.DMC_POS_Ctrl.Execute := TRUE;
		IF dmc_inputs.DMC_POS_Status.Busy THEN
			iMove := 20;
		END_IF
	20:
		IF NOT dmc_inputs.DMC_POS_Status.Busy THEN
			IF dmc_inputs.DMC_POS_Status.InTarget THEN
				iMove := 0;
			ELSE
				iMove :=99;
			END_IF
			dmc_outputs.DMC_POS_Ctrl.Execute := FALSE;
		END_IF
END_CASE
END_METHOD

PROPERTY PUBLIC Scale : real
GET
Scale := _scale;
END_GET
SET
_scale := Scale;
END_SET
END_PROPERTY

PROPERTY PUBLIC StartType : uint
GET
StartType := _startType;
END_GET
SET
_startType := StartType;
END_SET
END_PROPERTY

END_FUNCTION_BLOCK

// ---- Motion/StepperAxis/Ex70x7_DMC_Channel.TcPOU
FUNCTION_BLOCK Ex70x7_DMC_Channel
VAR_INPUT
END_VAR
VAR_OUTPUT
END_VAR
VAR
	ENCStatus AT%I* : StepperENCStatus;
	STMStatus AT%I* : StepperSTMStatus;
	POSStatus AT%I* : StepperPOSStatus;
	
	ENCControl AT%Q* : StepperENCControl;
	STMControl AT%Q* : StepperSTMControl;
	POSControl AT%Q* : StepperPOSControl;
	
	_InTarget : BOOL;
	
	State :(
		_00_mWait,
        _01_mReset,
        _02_mEnable,
		_06_mGotoPosition,
		_07_mStop,
		_08_mSetPosition,
		_09_RunAtExternalVelo,
		_10_Disable);
		
	tonHoldHigh				: ton;
END_VAR

CASE State OF
        _00_mWait : 
			;
        _01_mReset : 
			STMControl.Reset := TRUE;
			tonHoldHigh(in := TRUE, pt := T#500MS);
			IF tonHoldHigh.Q THEN
				STMControl.Reset := FALSE;
				IF STMStatus.Error = FALSE AND
					STMStatus.Warning = FALSE AND
					STMStatus.Ready = TRUE
				THEN
					State := _00_mWait;
					tonHoldHigh(in := FALSE, pt := T#500MS);
				END_IF
			END_IF
			
        _02_mEnable : 
			IF STMStatus.Error THEN				
				State := _01_mReset;
			ELSE
				STMControl.Enable := TRUE;			
			END_IF
			
		_06_mGotoPosition :
			POSControl.Execute := TRUE;
			_InTarget := FALSE;
			IF POSStatus.InTarget THEN
				State := _02_mEnable;
				POSControl.Execute := FALSE;
				_InTarget := TRUE;
			END_IF
			
		_07_mStop : 
			POSControl.Execute := FALSE;
			IF POSStatus.ReadyToExecute THEN	
				State := _02_mEnable;
			END_IF
			
		_08_mSetPosition :
			POSControl.Execute := TRUE;
			
			IF POSStatus.Calibrated THEN
				POSControl.Execute := FALSE;
				State := _02_mEnable;
			END_IF
			
		_09_RunAtExternalVelo :
			POSControl.Execute := TRUE;
			_InTarget := false;
			
		_10_Disable:
			STMControl.Enable := FALSE;
			State := _00_mWait;
		
			
END_CASE

PROPERTY ActualPosition : lreal
GET
ActualPosition := UDINT_TO_LREAL( POSStatus.ActualPosition)/8062.72;
END_GET
END_PROPERTY

PROPERTY ActualVelocity : int
GET
ActualVelocity := POSStatus.ActualVelocity;
END_GET
END_PROPERTY

METHOD CalibrateMotor : BOOL
VAR_INPUT
END_VAR
IF State = _02_mEnable THEN
	State := _08_mSetPosition;
	//POSControl.Velocity := REAL_TO_INT( Velocity*252);
	POSControl.StartType := StartType.Calibrate;
	//POSControl.TargetPosition := LREAL_TO_UDINT(Position*8062.72);
	//POSControl.TargetPosition := LREAL_TO_UDINT(Position*10);
END_IF
END_METHOD

METHOD Disable : BOOL
VAR_INPUT
END_VAR
IF STMStatus.Ready THEN
	State := _10_Disable;
END_IF
END_METHOD

METHOD Enable : BOOL
VAR_INPUT
END_VAR
IF STMStatus.ReadyToEnable THEN
	State := _02_mEnable;
END_IF
END_METHOD

METHOD GoToPosition : BOOL
VAR_INPUT
	Position : LREAL;
	Velocity : REAL;
END_VAR
IF State = _02_mEnable THEN
	State := _06_mGoToPosition;
	POSControl.Velocity := REAL_TO_INT( Velocity*252);
	POSControl.StartType := StartType.Absolute;
	POSControl.TargetPosition := LREAL_TO_UDINT(Position*8062.72);
END_IF
END_METHOD

PROPERTY InTarget : bool
GET
InTarget := _InTarget;
END_GET
END_PROPERTY

METHOD MoveAtVelocity : BOOL
VAR_INPUT
	Velocity : REAL;
END_VAR
IF State = _02_mEnable THEN
	State := _09_RunAtExternalVelo;
	POSControl.Velocity := REAL_TO_INT( Velocity*252);
	POSControl.StartType := StartType.VeloPositive;
END_IF
END_METHOD

PROPERTY Ready : bool
GET
Ready := STMStatus.Ready;
END_GET
END_PROPERTY

METHOD Reset : BOOL
VAR_INPUT
END_VAR
IF STMStatus.Error OR STMStatus.Warning OR POSStatus.Error THEN
	State := _01_mReset;
END_IF
END_METHOD

METHOD Stop : BOOL
VAR_INPUT
END_VAR
IF POSControl.Execute THEN
	State  := _07_mStop;
END_IF
END_METHOD

END_FUNCTION_BLOCK

// ---- Profibus/ProfibusDeviceBase.TcPOU
FUNCTION_BLOCK ProfibusDeviceBase
VAR_INPUT
END_VAR
VAR_OUTPUT
END_VAR
VAR
	DpState AT%I* : USINT;
	ExtDiagFlag at%i* : BOOL;
END_VAR

END_FUNCTION_BLOCK

// ---- Profibus/ProfibusMaster.TcPOU
FUNCTION_BLOCK ProfibusMaster
VAR_INPUT
END_VAR
VAR_OUTPUT
END_VAR
VAR
	Error AT%I* : USINT;
	ActualModulo AT%I* : USINT;
	DiagFlag AT%i* : BOOL;
END_VAR

END_FUNCTION_BLOCK

// ---- ProfiNet/ProfiNetDeviceBase.TcPOU
FUNCTION_BLOCK ProfiNetDeviceBase
VAR_INPUT
END_VAR
VAR_OUTPUT
END_VAR
VAR
	PnIoDeviceState AT%I* : UINT;
	PnIoDeviceDiag AT%i* : uint;
END_VAR

END_FUNCTION_BLOCK

// ---- ProfiNet/ProfiNetMaster.TcPOU
FUNCTION_BLOCK ProfiNetMaster
VAR_INPUT
END_VAR
VAR_OUTPUT
END_VAR
VAR
	DevState AT%I* : UINT;
	PnIoError AT%I* : UINT;
	PnIoDiag AT%i* : UINT;
END_VAR

END_FUNCTION_BLOCK
